// Swaps the parameters of two generic values.
FUNCTION F_SwapGenericsParameters
VAR_IN_OUT
	A : FsCommon.T_Generic; // Generic whose parameters will be swapped with B.
	B : FsCommon.T_Generic; // Generic whose parameters will be swapped with B.
END_VAR
VAR
	Tmp : FsCommon.T_Generic;
END_VAR

Tmp := A;
A 	:= B;
B 	:= Tmp;

END_FUNCTION

(* stored: Version 1.1.0.1
   POU F_SwapGenericsParameters: Id {57ec33c8-4605-086d-395f-e0dd044e32da}, SpecialFunc None *)
